// TIA Portal project "LineaContapezzi" (V20)

(* hardware
DEVICE "S7-1200 station_1"  S7-1200 Station
   slot 0: "Rack_0"  S7-1200 Rack  Rack  V1.0
   slot 1: "Playground_PLC"  CPU 1214C DC/DC/DC  6ES7 214-1AG40-0XB0  V4.7
   slot 3: "AQ 1x12BIT_1"  AQ1 signal board  6ES7 232-4HA30-0XB0  V1.0
*)

// ===== PLC "Playground_PLC"  CPU 1214C DC/DC/DC =====

VAR_GLOBAL   // PLC tag table "Default tag table"
   "P1" AT %M0.0 : Bool;
   "FC_TOT" AT %M0.1 : Bool;
   "BOTT_TOT" AT %MW1 : Int;
   "FC_MET" AT %M0.3 : Bool;
   "BOTT_MET" AT %MW2 : Int;
   "FC_PLS" AT %M0.5 : Bool;
   "BOTT_PLS" AT %MW3 : Int;
END_VAR

DATA_BLOCK "CONTABOTTIGLIE_TOT"   // DB1
{ S7_Optimized_Access := 'TRUE' }
VERSION : 0.1
// stored: InstanceOfName CONTABOTTIGLIE
"CONTABOTTIGLIE"
BEGIN
END_DATA_BLOCK

DATA_BLOCK "CONTABOTTIGLIE_PLS"   // DB2
{ S7_Optimized_Access := 'TRUE' }
VERSION : 0.1
// stored: InstanceOfName CONTABOTTIGLIE
"CONTABOTTIGLIE"
BEGIN
END_DATA_BLOCK

DATA_BLOCK "CONTABOTTIGLIE_MET"   // DB3
{ S7_Optimized_Access := 'TRUE' }
VERSION : 0.1
// stored: InstanceOfName CONTABOTTIGLIE
"CONTABOTTIGLIE"
BEGIN
END_DATA_BLOCK

FUNCTION_BLOCK "CONTABOTTIGLIE"   // FB1, LAD
{ S7_Optimized_Access := 'TRUE' }
VERSION : 0.1
   VAR_INPUT
      FOTOCELLULA : Bool;
   END_VAR
   VAR_OUTPUT
      PEZZI_CONTATI : Int;
   END_VAR
   VAR RETAIN
      IEC_Counter_0_Instance : CTU_INT;
   END_VAR
   VAR CONSTANT
      MAX_COUNT : Int := 9999;
   END_VAR
BEGIN

REGION Network 1
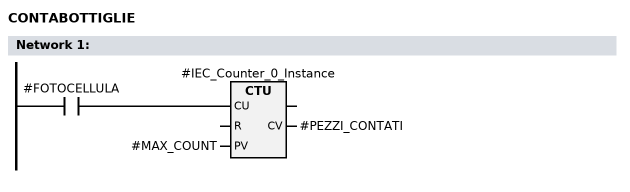
   #IEC_Counter_0_Instance(CU := #FOTOCELLULA, PV := #MAX_COUNT, CV => #PEZZI_CONTATI);   // CTU
END_REGION
END_FUNCTION_BLOCK

ORGANIZATION_BLOCK "Main"   // OB1, LAD, ProgramCycle
TITLE = "Main Program Sweep (Cycle)"
{ S7_Optimized_Access := 'TRUE' }
VERSION : 0.1
   VAR_INPUT
      Initial_Call : Bool;   // Initial call of this OB
      Remanence : Bool;   // =True, if remanent data are available
   END_VAR
   VAR_TEMP   // added for the SCL form of the ladder/FBD networks
      _w1 : Bool;
   END_VAR
BEGIN

REGION Network 1
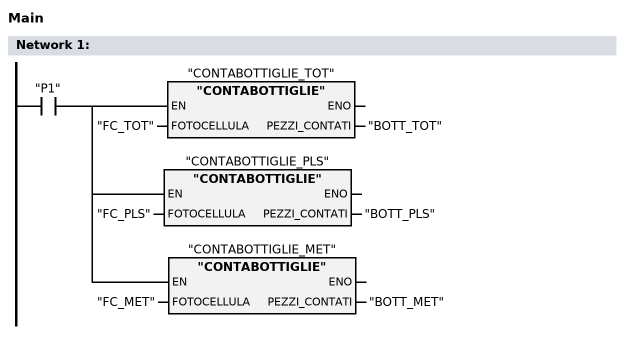
   RUNG wire#powerrail
      Contact( "P1" )
      wire#w1
      "CONTABOTTIGLIE_TOT"(FOTOCELLULA := "FC_TOT", PEZZI_CONTATI => "BOTT_TOT")
   END_RUNG
   RUNG wire#w1
      "CONTABOTTIGLIE_PLS"(FOTOCELLULA := "FC_PLS", PEZZI_CONTATI => "BOTT_PLS")
   END_RUNG
   RUNG wire#w1
      "CONTABOTTIGLIE_MET"(FOTOCELLULA := "FC_MET", PEZZI_CONTATI => "BOTT_MET")
   END_RUNG
   // the same network as SCL:
   #_w1 := "P1";
   IF #_w1 THEN
       "CONTABOTTIGLIE_TOT"(FOTOCELLULA := "FC_TOT", PEZZI_CONTATI => "BOTT_TOT");   // "CONTABOTTIGLIE"
       "CONTABOTTIGLIE_PLS"(FOTOCELLULA := "FC_PLS", PEZZI_CONTATI => "BOTT_PLS");   // "CONTABOTTIGLIE"
       "CONTABOTTIGLIE_MET"(FOTOCELLULA := "FC_MET", PEZZI_CONTATI => "BOTT_MET");   // "CONTABOTTIGLIE"
   END_IF;
END_REGION
END_ORGANIZATION_BLOCK